{attribute addProperty BoxType "EL1259-0000-0018"}
{attribute addProperty Id "CtrlAT %Q*Ctrl_8EDFA0AF3241OutputsAT %Q*Outputs_C23F921918623.2533Output_event_timeAT %Q*ARRAY[0 ..9] OF UDINT320400"}
{attribute addProperty CRC "1690710971"}
{attribute addProperty SizeInBites "538"}
{attribute addProperty SizeInBytes "67.25"}
TYPE MTO_Outputs_10x_Channel_6165A3A8 :
STRUCT
	{attribute addProperty Name "Ctrl"}
	Ctrl AT %Q* : Ctrl_8EDFA0AF;
	{attribute addProperty Name "Outputs"}
	Outputs AT %Q* : Outputs_C23F9219;
	{attribute addProperty Name "Output_event_time"}
	Output_event_time AT %Q* : ARRAY[0 ..9] OF UDINT;
END_STRUCT
END_TYPE

(* stored: Version 1.2.0.0, ProductVersion 3.1.4024.9
   DUT MTO_Outputs_10x_Channel_6165A3A8: Id {fc2277b4-b5d4-4ecc-890d-afd83596338f} *)
